// TIA Portal project "Paketband_2" (V20)

(* hardware
DEVICE "S7-300/ET200M-Station_1"  S7-300 station
   slot 0: "Profilschiene_0"  Rail  6ES7 390-1***0-0AA0
   slot 2: "PLC_1"  CPU 315-2 PN/DP  6ES7 315-2EH14-0AB0  V3.2.18
      slot 2: "PROFINET-Schnittstelle_1"  PN-IO
         slot 1: "Port_1"  Port
         slot 2: "Port_2"  Port
   slot 4: "DI 16x24VDC_1"  DI16 x 24VDC, interrupt  6ES7 321-7BH01-0AB0
   slot 5: "DO 8x24VDC/0.5A_1"  DO8 x 24VDC / 0.5A  6ES7 322-8BF00-0AB0
*)

// ===== PLC "PLC_1"  CPU 315-2 PN/DP =====

VAR_GLOBAL   // PLC tag table "Standard-Variablentabelle"
   "Förderband_an" AT %M1.2 : Bool;
   "Förderband_aus" AT %M1.3 : Bool;
   "NotAus_aktiv" AT %M1.1 : Bool;
   "Takt_100Hz" AT %M100.5 : Bool;
   "Anlage_ein" AT %M1.0 : Bool;
   "Paket_erkannt" AT %M1.4 : Bool;
   "Temp_1" AT %M0.0 : Bool;
   "Temp_2" AT %M0.1 : Bool;
END_VAR

VAR_GLOBAL   // PLC tag table "Eingänge"
   "S1" AT %E0.4 : Bool;   // Start-Taster
   "S2" AT %E0.5 : Bool;   // Stopp-Taster
   "S4" AT %E0.0 : Bool;   // Not-Aus Schalter
   "S0" AT %E0.1 : Bool;   // Betriebsschalter auf ein
   "S3" AT %E0.6 : Bool;   // Rücksetz-Taster
   "S5" AT %E1.0 : Bool;   // Wiedereinschalten Taster
   "1b1" AT %E1.1 : Bool;   // Lichttaster (Mitte)
   "2b1" AT %E1.2 : Bool;   // Lichttaster (Ende)
END_VAR

VAR_GLOBAL   // PLC tag table "Ausgänge"
   "S1_Licht" AT %A0.4 : Bool;   // Lampe des Start-Tasters
   "S2_Licht" AT %A0.5 : Bool;   // Lampe des Stopp-Tasters
   "M1" AT %A0.0 : Bool;   // Förderband
   "S3_Licht" AT %A0.6 : Bool;   // Lampe des Rücksetz-Tasters
   "H1" AT %A0.1 : Bool;   // Meldeleuchte (Grün)
   "H2" AT %A0.2 : Bool;   // Meldeleuchte (Gelb)
   "H3" AT %A0.3 : Bool;   // Meldeleuchte (Rot)
END_VAR

FUNCTION "Paketbandanlage" : Void   // FC1, FBD
{ S7_Optimized_Access := 'FALSE' }
VERSION : 0.1
   VAR_TEMP   // added for the SCL form of the ladder/FBD networks
      _w1 : Bool;
      _w2 : Bool;
   END_VAR
BEGIN

REGION Network 1: Paketbandsteuerung
   // Hinweis: Alle Schalter können nur benutzt werden, wenn die Anlage über den Betriebsschalter eingeschaltet wurde.
   // Das Paketband kann dann über S1 (Start-Taster) eingeschaltet werden bzw. durch S5 (Wiedereinschalten) und läuft dann dauerhaft. Über S2 (Stopp-Taster), 1b1 bzw. 2b1 (Lichttaster) wird das Paketband gestoppt. Der Stopp-Modus, kann durch den Start bzw. Wiedereinschalten deaktiviert werden.
   // Beide Modi (Start, Stopp) werden deaktiviert, sobald S4 (Not-Aus Schalter) aktiv ist.
   // Der Not-Aus-Modus kann nur über S3 (Rücksetz-Taster) deaktiviert werden.
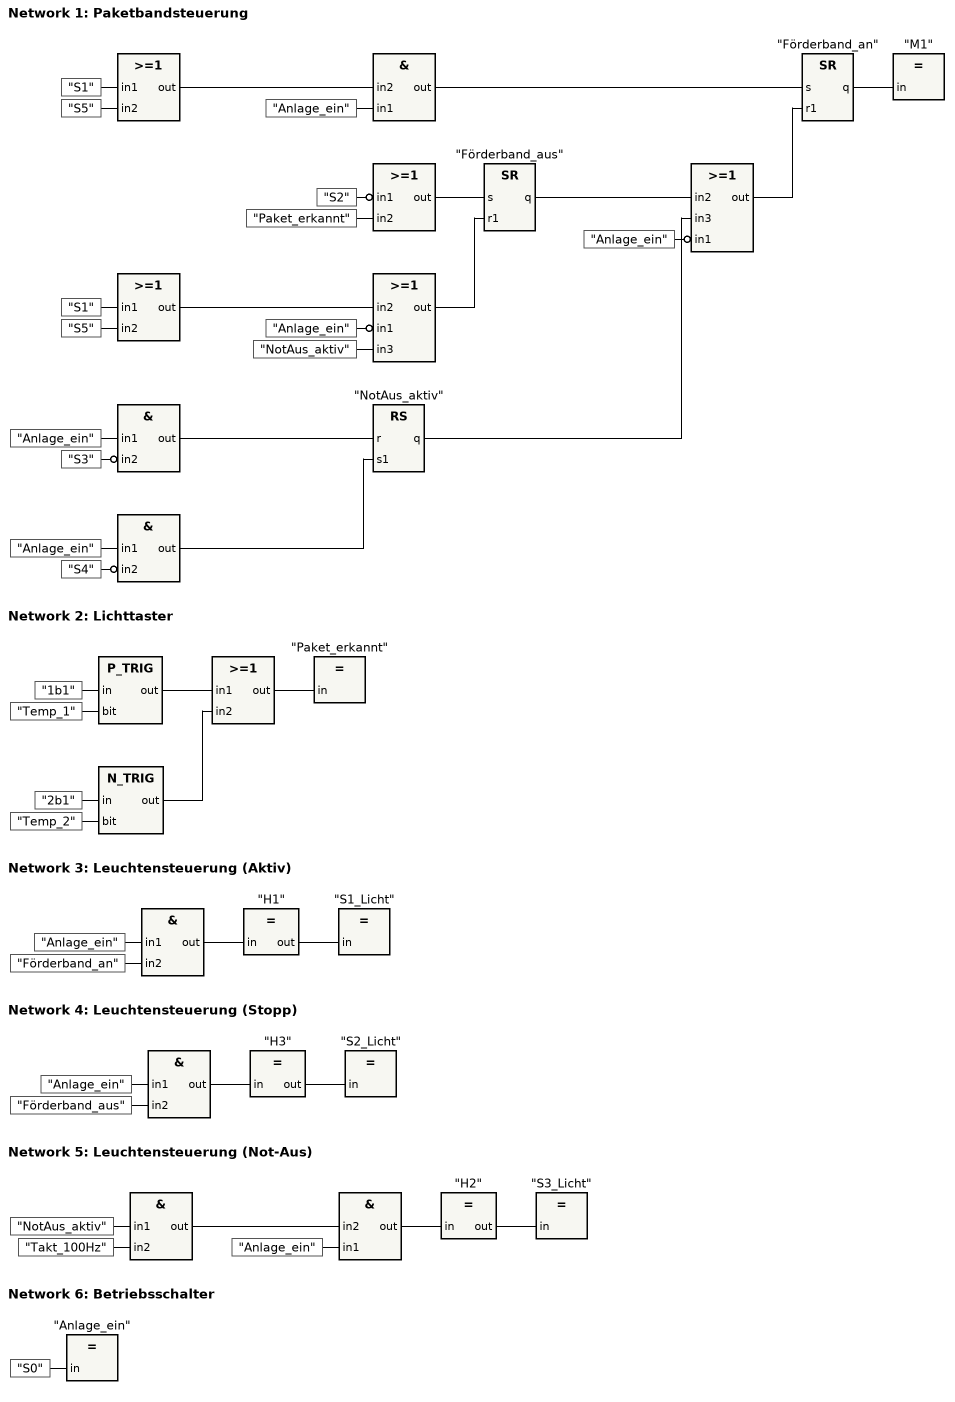
   IF NOT "S2" OR "Paket_erkannt" THEN
       "Förderband_aus" := TRUE;   // SR flip-flop
   END_IF;
   IF "S1" OR "S5" OR NOT "Anlage_ein" OR "NotAus_aktiv" THEN "Förderband_aus" := FALSE; END_IF;
   IF "Anlage_ein" AND NOT "S3" THEN
       "NotAus_aktiv" := FALSE;   // RS flip-flop
   END_IF;
   IF "Anlage_ein" AND NOT "S4" THEN "NotAus_aktiv" := TRUE; END_IF;
   IF ("S1" OR "S5") AND "Anlage_ein" THEN
       "Förderband_an" := TRUE;   // SR flip-flop
   END_IF;
   IF "Förderband_aus" OR "NotAus_aktiv" OR NOT "Anlage_ein" THEN "Förderband_an" := FALSE; END_IF;
   "M1" := "Förderband_an";
END_REGION

REGION Network 2: Lichttaster
   // Wenn 2b1 (der Lichttaster am Ende) oder 1b1 (Lichttaster in der Mitte) ein Paket erkennen, soll sofort bzw. verzögert das Band stehen bleiben.
   #_w1 := "1b1" AND NOT "Temp_1";   // rising edge
   "Temp_1" := "1b1";
   #_w2 := NOT "2b1" AND "Temp_2";   // falling edge
   "Temp_2" := "2b1";
   "Paket_erkannt" := #_w1 OR #_w2;
END_REGION

REGION Network 3: Leuchtensteuerung (Aktiv)
   // Wenn die Anlage ein ist und gestartet wurde, dann soll die Meldeleuchte und die Leuchte des Start-Tasters leuchten.
   "H1" := "Anlage_ein" AND "Förderband_an";
   "S1_Licht" := "H1";
END_REGION

REGION Network 4: Leuchtensteuerung (Stopp)
   // Wenn die Anlage ein ist, aber gestoppt wurde, dann soll die Meldeleuchte und die Leuchte des Stopp-Tasters leuchten.
   "H3" := "Anlage_ein" AND "Förderband_aus";
   "S2_Licht" := "H3";
END_REGION

REGION Network 5: Leuchtensteuerung (Not-Aus)
   // Wenn die Anlage ein ist und sich im Not-Aus befindet, dann soll die Meldeleuchte und die Leuchte des Rücksetz-Tasters blinken.
   "H2" := "NotAus_aktiv" AND "Takt_100Hz" AND "Anlage_ein";
   "S3_Licht" := "H2";
END_REGION

REGION Network 6: Betriebsschalter
   // Wenn der Betriebsschalter auf ein steht, sollen bestimmte Funktionsweisen möglich sein.
   "Anlage_ein" := "S0";
END_REGION
END_FUNCTION

ORGANIZATION_BLOCK "Main"   // OB1, FBD
TITLE = "Main Program Sweep (Cycle)"
{ S7_Optimized_Access := 'FALSE' }
VERSION : 0.1
   VAR_TEMP
      OB1_EV_CLASS : Byte;   // Bits 0-3 = 1 (Coming event), Bits 4-7 = 1 (Event class 1)
      OB1_SCAN_1 : Byte;   // 1 (Cold restart scan 1 of OB 1), 3 (Scan 2-n of OB 1)
      OB1_PRIORITY : Byte;   // Priority of OB Execution
      OB1_OB_NUMBR : Byte;   // 1 (Organization block 1, OB1)
      OB1_RESERVED_1 : Byte;   // Reserved for system
      OB1_RESERVED_2 : Byte;   // Reserved for system
      OB1_PREV_CYCLE : Int;   // Cycle time of previous OB1 scan (milliseconds)
      OB1_MIN_CYCLE : Int;   // Minimum cycle time of OB1 (milliseconds)
      OB1_MAX_CYCLE : Int;   // Maximum cycle time of OB1 (milliseconds)
      OB1_DATE_TIME : Date_And_Time;   // Date and time OB1 started
   END_VAR
BEGIN

REGION Network 1
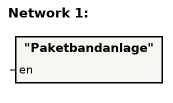
   "Paketbandanlage"();
END_REGION
END_ORGANIZATION_BLOCK